TYPE ST_Message :
STRUCT
  eType         : e_MessageType;
  eDevice       : e_Device;
  eSubdevice    : e_SubDevice;
  {attribute 'displaymode':='hex'}
  iErrorNumber  : LINT;
  tTime         : STRING(24);
  sText         : STRING(127);
END_STRUCT
END_TYPE

(* stored: Version 1.1.0.1
   DUT ST_Message: Id {42213b33-b0ef-40c6-a9c4-0e691a7c5cd8} *)
